// TIA Portal V17 export
// export: Created 2023-02-25T15:48:30.3158817Z, ExportSetting WithDefaults, DisplayName Totally Integrated Automation Portal, DisplayVersion V17, DisplayName TIA Portal Openness, DisplayVersion V17, DisplayName TIA Portal Version Control Interface, DisplayVersion V17, DisplayName TIA Portal Test Suite Advanced, DisplayVersion V17, DisplayName STEP 7 Professional, DisplayVersion V17, DisplayName SIMATIC Energy Suite, DisplayVersion V17, DisplayName STEP 7 Safety, DisplayVersion V17, DisplayName WinCC Professional, DisplayVersion V17
DATA_BLOCK "LOG_ManualModule_DB"   // DB12
VERSION : 0.1
// stored: AutoNumber true, InstanceOfName LOG_ManualModule, InstanceOfType FB
"LOG_ManualModule"
   // VAR_INPUT
   //    StartLine : Bool;
   //    StopLine : Bool;
   //    ModeManual : Bool;
   //    ButtonAction : Bool;
   // END_VAR
   // VAR_OUTPUT
   //    StartAction : Bool;
   // END_VAR
   // VAR RETAIN
   //    IEC_Counter_0_Instance { ExternalAccessible := 'False'; ExternalVisible := 'False'; ExternalWritable := 'False'} : CTU_INT;
   // END_VAR
   // VAR
   //    P_ButtonAction : Bool;
   //    CV : Int;
   //    Reset : Bool;
   // END_VAR
BEGIN
END_DATA_BLOCK
